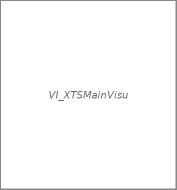
VISUALIZATION MAIN_VISU  // 177x190
    Frame (0,0 177x190)
        shows VI_XTSMainVisu(xts := XTS_PRG.fbXTSSystem)
END_VISUALIZATION

(* stored: Version 1.1.0.1, ProductVersion 3.1.4024.11
   Visu MAIN_VISU: Id {b6f6d5f1-9655-4e79-9d72-2bc06c42051f} *)
